// TIA Portal V20 export
FUNCTION_BLOCK "FB_DecodChannels"   // FB405, SCL
{ S7_Optimized_Access := 'TRUE' }
// stored: AutoNumber false, MemoryReserve 100, SetENOAutomatically false
   VAR DB_SPECIFIC
      sChan1IsDisplayed : Bool;
      sChan2IsDisplayed : Bool;
      sChan3IsDisplayed : Bool;
      sChan4IsDisplayed : Bool;
   END_VAR
   VAR CONSTANT
      CH00 : Byte := 0;
      CH01 : Byte := 1;
      CH02 : Byte := 2;
      CH03 : Byte := 3;
      CH04 : Byte := 4;
   END_VAR
BEGIN
   REGION Description header 
       //==================================================================================
       // POSALUX Swiss SA / (C) Copyright 2025
       //----------------------------------------------------------------------------------
       // Title: FB_DecodChannels
       // Comment/Function: Indication of the displayed channel according to the
       //                   current channel number
       // Author: Fabien WALDT
       // Engineering: TIA Portal v17
       //----------------------------------------------------------------------------------
       // Change log table:
       // Version  | Date     | Expert in charge | Changes applied
       // ---------|----------|------------------|-----------------------------------------
       // 00.00.01 | 20250505 | WFA              | First released version
       // =================================================================================
   END_REGION

   REGION Channel decoding
       CASE "LBP_HMI".E_Chan OF
           #CH00:
               #sChan1IsDisplayed := 0;
               #sChan2IsDisplayed := 0;
               #sChan3IsDisplayed := 0;
               #sChan4IsDisplayed := 0;
           #CH01:
               #sChan1IsDisplayed := 1;
               #sChan2IsDisplayed := 0;
               #sChan3IsDisplayed := 0;
               #sChan4IsDisplayed := 0;
           #CH02:
               #sChan1IsDisplayed := 0;
               #sChan2IsDisplayed := 1;
               #sChan3IsDisplayed := 0;
               #sChan4IsDisplayed := 0;
           #CH03:
               #sChan1IsDisplayed := 0;
               #sChan2IsDisplayed := 0;
               #sChan3IsDisplayed := 1;
               #sChan4IsDisplayed := 0;
           #CH04:
               #sChan1IsDisplayed := 0;
               #sChan2IsDisplayed := 0;
               #sChan3IsDisplayed := 0;
               #sChan4IsDisplayed := 1;
           ELSE
               #sChan1IsDisplayed := 0;
               #sChan2IsDisplayed := 0;
               #sChan3IsDisplayed := 0;
               #sChan4IsDisplayed := 0;
       END_CASE;
   END_REGION
END_FUNCTION_BLOCK
